(*********************************** G.D S.p.A. - Technical Department ***********************************
============= PROGRAM INFO ============
FOLDER:             TBD
MACHINES INVOLVED:  TBD 

============= DESCRIPTION =============
Machine declaration

============= REVISIONS ===============
Date		Version	 	Author      	Description             
----------	-------		------------  	--------------------------------------------
2019/03/27 	0000.00	 	CEC 			Creation of the PRG

**********************************************************************************************************)

TYPE csp_customerInterfaces_casePackerStRate :
STRUCT
	
	Target:			INT;				(*$H_R desc := Target rate in Pods/minute; $*)
	Actual:			INT;				(*$H_R desc := REAL-TIME rate in Pods/minute; $*)
															
END_STRUCT
END_TYPE

(* stored: Version 1.1.0.1, ProductVersion 3.1.4024.3
   DUT csp_customerInterfaces_casePackerStRate: Id {a09540b4-31a9-4e83-8ea1-18688a25d293} *)
